// TIA Portal V21 export
TYPE "Std_Lpf"
   STRUCT
      Setpoint : Real;
      FattoreFiltro : Real;
      ValoreFiltrato : Real;
   END_STRUCT;
END_TYPE
